// TIA Portal project "gaugungStation" (V17)

(* hardware
DEVICE "S7-1200 station_1"  S7-1200 Station
   slot 0: "Rack_0"  S7-1200 Rack  Rack  V1.0
   slot 1: "PLC_1"  CPU 1214C DC/DC/DC  6ES7 214-1AG40-0XB0  V4.4
DEVICE "ET 200SP station_1"  ET 200SP-Station
   slot 0: "Rack_0"  Rack  6ES5 710-8MAx1
   slot 0: "IO device_1"  IM 155-6 PN/2 HF  6ES7 155-6AU01-0CN0  V4.2
   slot 1: "DI 8x24VDC HF_1"  DI 8x24VDC HF  6ES7 131-6BF00-0CA0  V2.0
      slot 1: "DI 8x24VDC HF_1"  DI 8x24VDC HF
   slot 2: "DI 8x24VDC HF_2"  DI 8x24VDC HF  6ES7 131-6BF00-0CA0  V2.0
      slot 1: "DI 8x24VDC HF_2"  DI 8x24VDC HF
   slot 3: "DI 8x24VDC HF_3"  DI 8x24VDC HF  6ES7 131-6BF00-0CA0  V2.0
      slot 1: "DI 8x24VDC HF_3"  DI 8x24VDC HF
   slot 4: "DQ 8x24VDC/0.5A HF_1"  DQ 8x24VDC/0.5A HF  6ES7 132-6BF00-0CA0  V2.0
      slot 1: "DQ 8x24VDC/0.5A HF_1"  DQ 8x24VDC/0.5A HF
   slot 5: "DQ 8x24VDC/0.5A HF_2"  DQ 8x24VDC/0.5A HF  6ES7 132-6BF00-0CA0  V2.0
      slot 1: "DQ 8x24VDC/0.5A HF_2"  DQ 8x24VDC/0.5A HF
   slot 6: "Server module_1"  Server module  6ES7 193-6PA00-0AA0  V1.1
      slot 1: "Server module_1"  Server module
   slot 127: "BA 2xRJ45"  BA 2xRJ45  6ES7 193-6AR00-0AA0  V0.0
      slot 1: "Port_1"  X1 P1 R  6ES7 193-6AR00-0AA0  V0.0
      slot 2: "Port_2"  X1 P2 R  6ES7 193-6AR00-0AA0  V0.0
DEVICE "SCALANCE X005"  SCALANCE X-Station
   slot 0: "SCALANCE X rack"  Rail
   slot 0: "Switch_1"  6GK5 005-0BA00-1AB2  V1.0
*)

// ===== PLC "PLC_1"  CPU 1214C DC/DC/DC =====

VAR_GLOBAL   // PLC tag table "Default tag table"
   "sysRun" AT %M0.0 : Bool;
   "height okay" AT %M0.1 : Bool;
   "heightNotOkay" AT %M0.2 : Bool;
   "wrongOrienation" AT %M0.3 : Bool;
   "correctOrientation" AT %M0.4 : Bool;
   "endReject" AT %M0.5 : Bool;
   "endTransfer" AT %M0.6 : Bool;
   "motor forward check" AT %M0.7 : Bool;
   "loop" AT %M1.0 : Bool;
   "initiation of the process after rejection" AT %M1.1 : Bool;
   "initiate process after transfer" AT %M1.2 : Bool;
   "step 1" AT %M1.3 : Bool;
   "step2" AT %M1.4 : Bool;
   "step 3" AT %M1.5 : Bool;
   "step 4" AT %M1.6 : Bool;
   "step 5" AT %M1.7 : Bool;
   "step 6" AT %M2.0 : Bool;
   "step 7" AT %M2.1 : Bool;
   "step 8" AT %M2.2 : Bool;
   "transferCylinderExtendedManually" AT %M2.3 : Bool;
   "Tag_1" AT %M10.0 : Bool;
   "Tag_2" AT %M102.1 : Bool;
   "Tag_3" AT %M102.7 : Bool;
   "Tag_4" AT %M201.0 : Bool;
   "resetMode" AT %M200.0 : Bool;
   "Tag_6" AT %M200.5 : Bool;
   "heightMeasured" AT %M203.4 : Bool;
END_VAR

VAR_GLOBAL   // PLC tag table "OurInputsAndOutputs"
   "Start button" AT %I0.0 : Bool;
   "Stop button" AT %I0.1 : Bool;
   "emergency stop" AT %I0.2 : Bool;
   "output power on" AT %I0.3 : Bool;
   "input 1 from previous station" AT %I0.4 : Bool;
   "input 2 from previous station" AT %I0.5 : Bool;
   "input 1 from next station" AT %I0.6 : Bool;
   "input 2 from next station" AT %I0.7 : Bool;
   "reset switch" AT %I1.0 : Bool;
   "auto switch" AT %I1.1 : Bool;
   "reject cylinder 3A retracted" AT %I1.2 : Bool;
   "reject cylinder 3A extended" AT %I1.3 : Bool;
   "transfer cylinder 1A retracted" AT %I1.4 : Bool;
   "transfer cylinder 1A extended" AT %I1.5 : Bool;
   "traverse in end of travel position" AT %I4.6 : Bool;
   "traverse in start of travel position" AT %I4.7 : Bool;
   "part in height measuring position" AT %I2.0 : Bool;
   "part height reading" AT %I2.1 : Bool;
   "port not detected" AT %I2.2 : Bool;
   "automatic ON lamp" AT %Q0.0 : Bool;
   "output 1 to previous station" AT %Q0.1 : Bool;
   "output 2 to previous sation" AT %Q0.2 : Bool;
   "output 1 to next station" AT %Q0.3 : Bool;
   "output 2 to next station" AT %Q0.4 : Bool;
   "extend reject cylinder 3A" AT %Q0.5 : Bool;
   "extend transfer cylinder 1A" AT %Q0.6 : Bool;
   "retract transfer cylinder 1A" AT %Q0.7 : Bool;
   "motor starter contactor(forward)" AT %Q1.0 : Bool;
   "motor starter contactor(revrese)" AT %Q1.1 : Bool;
   "extend lift cylinder 2A" AT %Q3.1 : Bool;
END_VAR

// folder: System blocks/Program resources

DATA_BLOCK "timer3"   // DB1
{ S7_Optimized_Access := 'TRUE' }
AUTHOR : Simatic
FAMILY : IEC
NAME : IEC_TMR
VERSION : 1.0
// stored: InstanceOfName IEC_TIMER
"IEC_TIMER"
BEGIN
END_DATA_BLOCK

DATA_BLOCK "timer8"   // DB2
{ S7_Optimized_Access := 'TRUE' }
AUTHOR : Simatic
FAMILY : IEC
NAME : IEC_TMR
VERSION : 1.0
// stored: InstanceOfName IEC_TIMER
"IEC_TIMER"
BEGIN
END_DATA_BLOCK

DATA_BLOCK "timer20"   // DB3
{ S7_Optimized_Access := 'TRUE' }
AUTHOR : Simatic
FAMILY : IEC
NAME : IEC_TMR
VERSION : 1.0
// stored: InstanceOfName IEC_TIMER
"IEC_TIMER"
BEGIN
END_DATA_BLOCK

DATA_BLOCK "timer7"   // DB4
{ S7_Optimized_Access := 'TRUE' }
AUTHOR : Simatic
FAMILY : IEC
NAME : IEC_TMR
VERSION : 1.0
// stored: InstanceOfName IEC_TIMER
"IEC_TIMER"
BEGIN
END_DATA_BLOCK

DATA_BLOCK "timer9"   // DB5
{ S7_Optimized_Access := 'TRUE' }
AUTHOR : Simatic
FAMILY : IEC
NAME : IEC_TMR
VERSION : 1.0
// stored: InstanceOfName IEC_TIMER
"IEC_TIMER"
BEGIN
END_DATA_BLOCK

DATA_BLOCK "timer34"   // DB6
{ S7_Optimized_Access := 'TRUE' }
AUTHOR : Simatic
FAMILY : IEC
NAME : IEC_TMR
VERSION : 1.0
// stored: InstanceOfName IEC_TIMER
"IEC_TIMER"
BEGIN
END_DATA_BLOCK

// folder: (top level)

ORGANIZATION_BLOCK "Main"   // OB1, LAD, ProgramCycle
TITLE = "Main Program Sweep (Cycle)"
{ S7_Optimized_Access := 'TRUE' }
VERSION : 0.1
   VAR_INPUT
      Initial_Call : Bool;   // Initial call of this OB
      Remanence : Bool;   // =True, if remanent data are available
   END_VAR
   VAR_TEMP   // added for the SCL form of the ladder/FBD networks
      _w1 : Bool;
      _w2 : Bool;
      _w3 : Bool;
   END_VAR
BEGIN

REGION Network 1: start condition
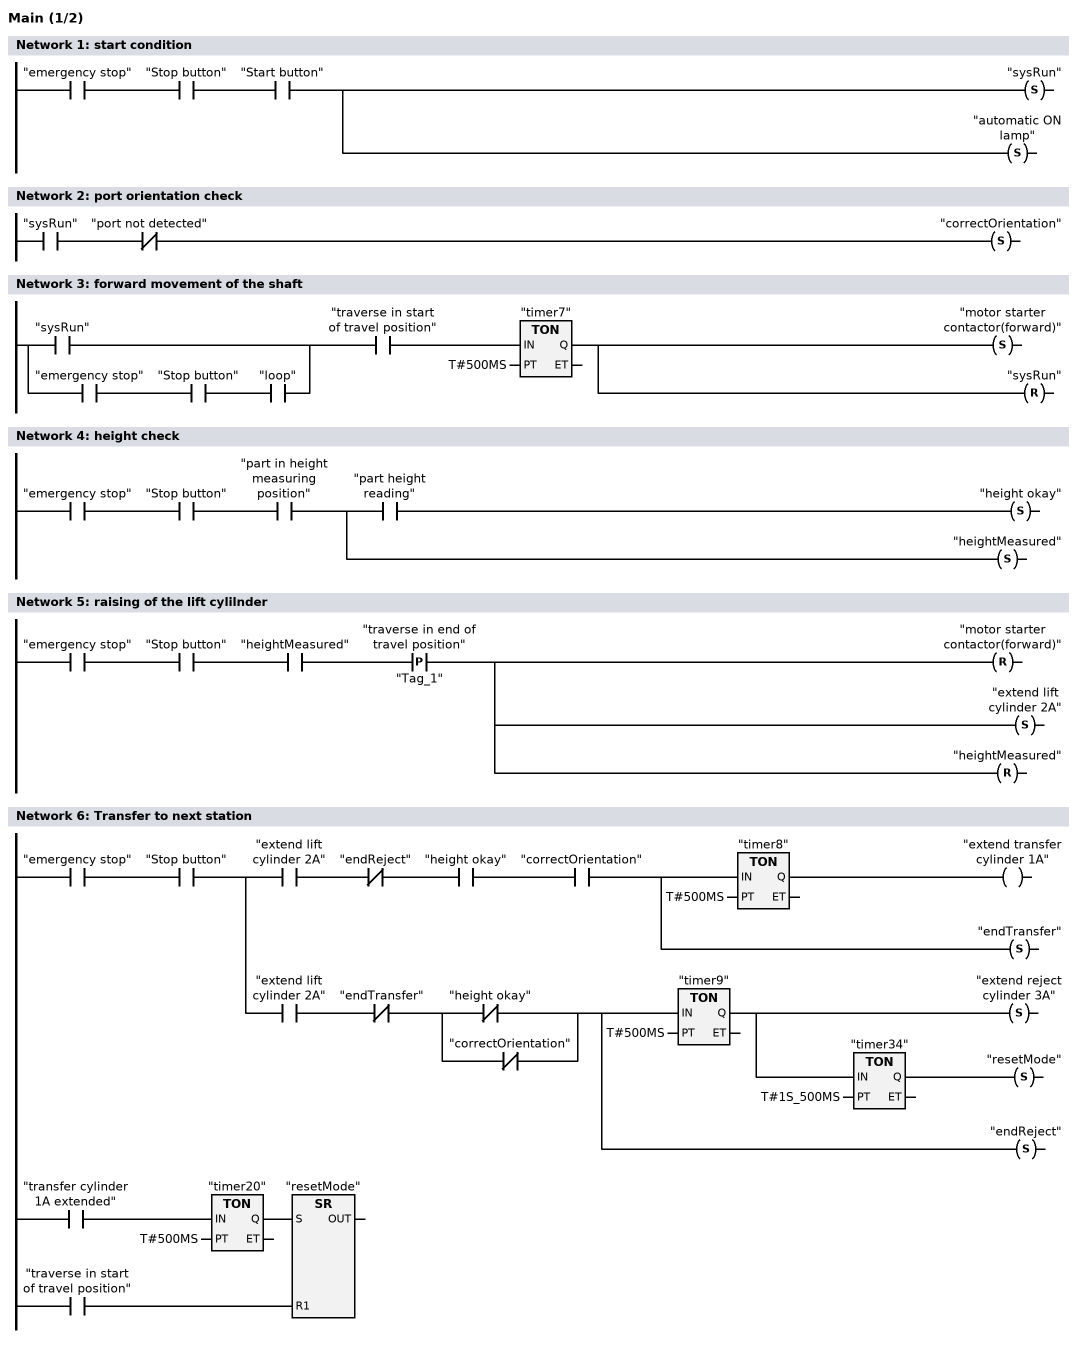
   RUNG wire#powerrail
      Contact( "emergency stop" )
      Contact( "Stop button" )
      Contact( "Start button" )
      wire#w1
      S_Coil( "sysRun" )
   END_RUNG
   RUNG wire#w1
      S_Coil( "automatic ON lamp" )
   END_RUNG
   // the same network as SCL:
   IF "emergency stop" AND "Stop button" AND "Start button" THEN
       "sysRun" := TRUE;
       "automatic ON lamp" := TRUE;
   END_IF;
END_REGION

REGION Network 2: port orientation check
   RUNG wire#powerrail
      Contact( "sysRun" )
      I_Contact( "port not detected" )
      S_Coil( "correctOrientation" )
   END_RUNG
   // the same network as SCL:
   IF "sysRun" AND NOT "port not detected" THEN "correctOrientation" := TRUE; END_IF;
END_REGION

REGION Network 3: forward movement of the shaft
   "timer7".TON(IN := ("sysRun" OR ("emergency stop" AND "Stop button" AND "loop")) AND "traverse in start of travel position",
                PT := T#500MS);
   IF "timer7".Q THEN
       "motor starter contactor(forward)" := TRUE;
       "sysRun" := FALSE;
   END_IF;
END_REGION

REGION Network 4: height check
   RUNG wire#powerrail
      Contact( "emergency stop" )
      Contact( "Stop button" )
      Contact( "part in height measuring position" )
      wire#w1
      Contact( "part height reading" )
      S_Coil( "height okay" )
   END_RUNG
   RUNG wire#w1
      S_Coil( "heightMeasured" )
   END_RUNG
   // the same network as SCL:
   #_w1 := "emergency stop" AND "Stop button" AND "part in height measuring position";
   IF #_w1 AND "part height reading" THEN "height okay" := TRUE; END_IF;
   IF #_w1 THEN "heightMeasured" := TRUE; END_IF;
END_REGION

REGION Network 5: raising of the lift cylilnder
   RUNG wire#powerrail
      Contact( "emergency stop" )
      Contact( "Stop button" )
      Contact( "heightMeasured" )
      P_Contact(operand := "traverse in end of travel position", bit := "Tag_1")
      wire#w1
      R_Coil( "motor starter contactor(forward)" )
   END_RUNG
   RUNG wire#w1
      S_Coil( "extend lift cylinder 2A" )
   END_RUNG
   RUNG wire#w1
      R_Coil( "heightMeasured" )
   END_RUNG
   // the same network as SCL:
   #_w1 := "emergency stop" AND "Stop button" AND "heightMeasured" AND "traverse in end of travel position" AND NOT "Tag_1";   // rising edge of "traverse in end of travel position"
   "Tag_1" := "traverse in end of travel position";
   IF #_w1 THEN
       "motor starter contactor(forward)" := FALSE;
       "extend lift cylinder 2A" := TRUE;
       "heightMeasured" := FALSE;
   END_IF;
END_REGION

REGION Network 6: Transfer to next station
   #_w1 := "emergency stop" AND "Stop button";
   #_w2 := #_w1 AND "extend lift cylinder 2A" AND NOT "endReject" AND "height okay" AND "correctOrientation";
   "timer8".TON(IN := #_w2, PT := T#500MS);
   "extend transfer cylinder 1A" := "timer8".Q;
   IF #_w2 THEN "endTransfer" := TRUE; END_IF;
   #_w3 := #_w1 AND "extend lift cylinder 2A" AND NOT "endTransfer" AND (NOT "height okay" OR NOT "correctOrientation");
   "timer9".TON(IN := #_w3, PT := T#500MS);
   IF "timer9".Q THEN "extend reject cylinder 3A" := TRUE; END_IF;
   "timer34".TON(IN := "timer9".Q, PT := T#1S_500MS);
   IF "timer34".Q THEN "resetMode" := TRUE; END_IF;
   IF #_w3 THEN "endReject" := TRUE; END_IF;
   "timer20".TON(IN := "transfer cylinder 1A extended", PT := T#500MS);
   IF "timer20".Q THEN
       "resetMode" := TRUE;   // SR flip-flop
   END_IF;
   IF "traverse in start of travel position" THEN "resetMode" := FALSE; END_IF;
END_REGION

REGION Network 7: Reset action
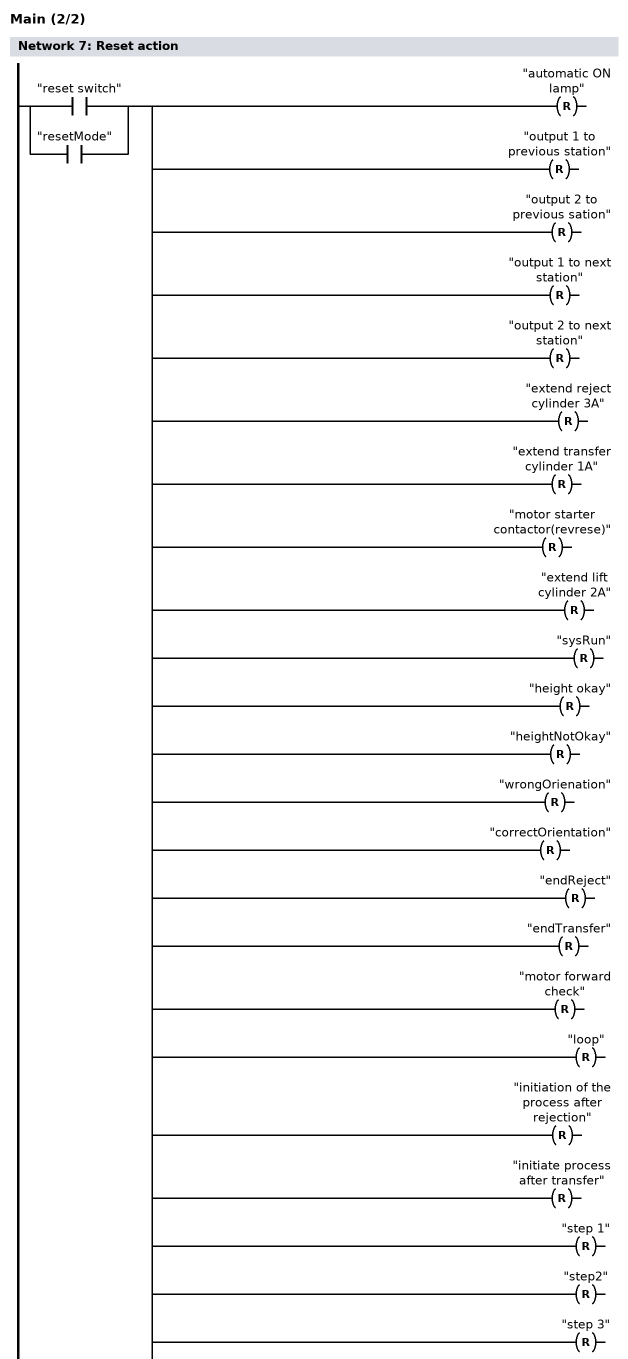
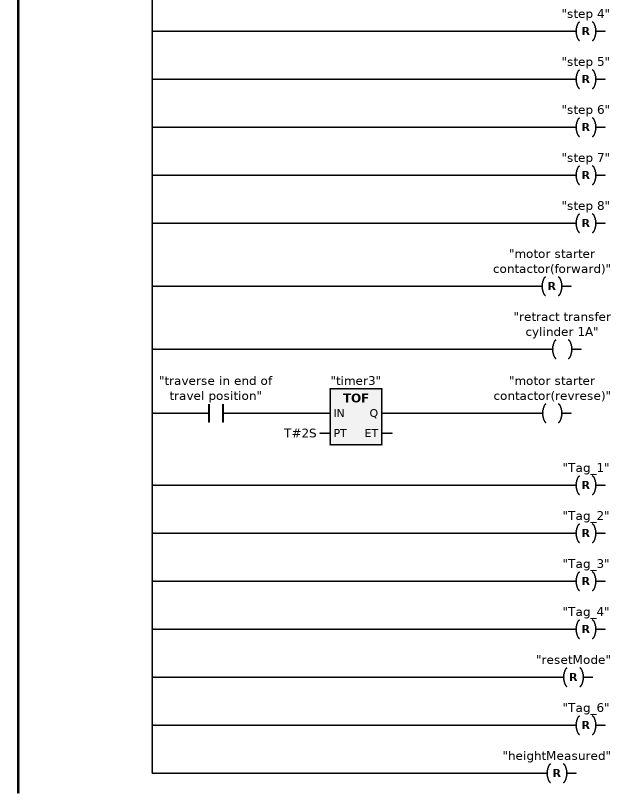
   #_w1 := "reset switch" OR "resetMode";
   IF #_w1 THEN
       "automatic ON lamp" := FALSE;
       "output 1 to previous station" := FALSE;
       "output 2 to previous sation" := FALSE;
       "output 1 to next station" := FALSE;
       "output 2 to next station" := FALSE;
       "extend reject cylinder 3A" := FALSE;
       "extend transfer cylinder 1A" := FALSE;
       "motor starter contactor(revrese)" := FALSE;
       "extend lift cylinder 2A" := FALSE;
       "sysRun" := FALSE;
       "height okay" := FALSE;
       "heightNotOkay" := FALSE;
       "wrongOrienation" := FALSE;
       "correctOrientation" := FALSE;
       "endReject" := FALSE;
       "endTransfer" := FALSE;
       "motor forward check" := FALSE;
       "loop" := FALSE;
       "initiation of the process after rejection" := FALSE;
       "initiate process after transfer" := FALSE;
       "step 1" := FALSE;
       "step2" := FALSE;
       "step 3" := FALSE;
       "step 4" := FALSE;
       "step 5" := FALSE;
       "step 6" := FALSE;
       "step 7" := FALSE;
       "step 8" := FALSE;
       "motor starter contactor(forward)" := FALSE;
   END_IF;
   "retract transfer cylinder 1A" := #_w1;
   "timer3".TOF(IN := #_w1 AND "traverse in end of travel position", PT := T#2S);
   "motor starter contactor(revrese)" := "timer3".Q;
   IF #_w1 THEN
       "Tag_1" := FALSE;
       "Tag_2" := FALSE;
       "Tag_3" := FALSE;
       "Tag_4" := FALSE;
       "resetMode" := FALSE;
       "Tag_6" := FALSE;
       "heightMeasured" := FALSE;
   END_IF;
END_REGION
END_ORGANIZATION_BLOCK